INTERFACE I_BINARY_SWITCH_SENS EXTENDS I_BINARY_SWITCH

METHOD M_START_SENS : BOOL
VAR_INPUT
	bState: BOOL;
	tDelay: TIME;
	eEventType: ENUM_EVENT_TYPE;
END_VAR
END_METHOD

METHOD M_STOP_SENS : BOOL
VAR_INPUT
END_VAR
END_METHOD

PROPERTY P_STATE_SENS : BOOL
GET
END_GET
END_PROPERTY

END_INTERFACE

(* stored: Version 1.1.0.1, ProductVersion 3.1.4024.9
   Itf I_BINARY_SWITCH_SENS: Id {b1dbad1d-3708-415c-b469-8ec427ec4d9f}
   Method M_START_SENS: Id {b2ba339f-8d1d-48a7-b231-24a35844b9c5}
   Method M_STOP_SENS: Id {1eb73ef8-d947-4886-b3b8-03d6a0260319}
   Property P_STATE_SENS: Id {ae4b5a92-877c-4476-9330-45d411ff13f4}
   Get Get: Id {8fd3c4d2-13e8-4b0c-bab3-4198798b1d11} *)
